FUNCTION_BLOCK FB_GGO
VAR_IN_OUT
	iq_astGauges: ARRAY[0..gc_iSizeOfGGOArray] OF ST_VG;
	iq_axHV_RO: ARRAY[0..gc_iSizeOfGGOArray] OF BOOL;
END_VAR
VAR_INPUT
	i_iIndex: INT;
END_VAR
VAR

	stPG: ST_VG;
	stVG: ST_VG;
	//index for associated pirani
	wPG : WORD;

	
	// FBs
	fb903	:	FB_903;
	fb907	:	FB_907;
	fb909	:	FB_909;
	fb925	:	FB_925;
	fbGCM	:	FB_GCM;
	
END_VAR

(* This function block is used to calculate the pressure from the analog input voltage and to provide protection and automatic turn on of ion gauges.
 It also manages the turn on fo the AT_VAC boolean, and checks to make sure the pressure is good *)

(* Full-scale pressure conversion factor *)

(* Real-value voltage calculation *)
(* Generic expression for pressure in the MKS systems

P = 10^(V/0.6-12)

722B = 0
903 = 1
907 = 2
909 = 3
925 = 4

*)

(* Make a copy of gauge at index*)
stVG := iq_astGauges[LIMIT(0 ,i_iIndex, gc_iSizeOfGGOArray)];

(* Check that it is an ion gauge *)
IF stVG.eTYPE = Gauge_Type.IG903 OR stVG.eTYPE = Gauge_Type.IG909 THEN

(* Check that Associated Gauge is within index*)
	IF WORD_TO_INT(stVG.wPG) <= gc_iSizeOfGGOArray THEN
		(* Check pressure gauge type before assignment *)
		(* Add high pressure gauge types here *)
		IF iq_astGauges[stVG.wPG].eTYPE = PG722B OR //722B
		iq_astGauges[stVG.wPG].eTYPE = PG907 OR //907
		iq_astGauges[stVG.wPG].eTYPE = PG925 THEN //925
			stPG := iq_astGauges[stVG.wPG];  (* Copy associated pirani gauge number to local variable *)
		ELSE //Default to allow the IG to turn on, this allows someone to set the PG to another IG and turn the gauge on whenever they want
			stPG.rPRESS := 1E-3;
			stPG.xPRESS_OK := TRUE;
		END_IF
	
	END_IF
END_IF

(* Evaluate each Gauge pressure based on eTYPE*)
CASE iq_astGauges[i_iIndex].eTYPE OF
	
	//Baratron Gauge
	PG722B:
		fbGCM(VG:=iq_astGauges[i_iIndex]);
		
	//Cold Cathode
	Gauge_Type.IG903:
		fb903(IG:=iq_astGauges[i_iIndex], PG:=iq_astGauges[wPG]);
		
	//Pirani Gauge	
	PG907:
		fb907(PG:=iq_astGauges[i_iIndex]);
		
	//Hot Cathode	
	Gauge_Type.IG909:
		fb909(IG:=iq_astGauges[i_iIndex], PG:=iq_astGauges[wPG]);
		
	//MicroPirani Gauge	
	PG925:
		fb925(VG:=iq_astGauges[i_iIndex]);
	ELSE
		(* Now, since we don't know what gauge type we're dealing with, we want 
		to make sure to reset all the gauge parameters, otherwise we may be 
		left with stale information *)
	stVG.rPRESS := 760;
	stVG.xAT_VAC := FALSE;
	stVG.xPRESS_OK := FALSE;
	stVG.xHV_SW := FALSE;
		
END_CASE

(* reAssign "HV On" back into High Voltage Array*)
iq_axHV_RO[LIMIT(0,WORD_TO_INT(stVG.wHV_RO),gc_iSizeOfGGOArray)]:=stVG.xHV_DIS;

END_FUNCTION_BLOCK

(* stored: Version 1.1.0.1, ProductVersion 3.1.4022.18
   POU FB_GGO: Id {10b35b2a-0339-4871-a987-1f7d7e8bc93e}, SpecialFunc None *)
